Yaskawa INFORM job: SIDE-B-CLAMP.JBI

/JOB
//NAME SIDE-B-CLAMP
///FOLDERNAME CLAMPUNCLAMP
//POS
///NPOS 0,0,0,0,0,0
//INST
///DATE 2021/10/04 12:18
///ATTR SC,RW
NOP
'********************************
'CLOSE CLAMP
'SIDE-B ARW CELL#2
'********************************
SET B099 0
'**CLOSE CLAMP**
DOUT OT#(169) OFF
DOUT OT#(170) ON
WAIT IN#(157)=ON T=3.00
JUMP *QUIT IF IN#(157)=OFF
'**CLAMPING COMPLETE**
SET B099 1
*QUIT
END
